// TIA Portal V19 export
TYPE "TMeasuring_Alarms"
// stored: Access Published
   STRUCT
      TOMeasuring : Bool;   // Alarm in technology object
      MCFunction : Bool;   // Alarm of MC function
      TimeOutActivation : Bool;   // Time out activation of measuring input
   END_STRUCT;
END_TYPE
